(* IEC 61131-3 sources: matiec/tests/upstream_fixes, 6 files *)

(* ---- array_initializer_overflow.st ---- *)
(* Regression test for c73c55d (beremiz/matiec): too many initial values for
 * an array used to reach generate_c_vardecl.cc and hit an internal compiler
 * error instead of being caught in stage 3.
 *
 * c73c55d alone is not enough: its check reads symbol->datatype off the
 * array_initial_elements_list_c node, which is only ever set by 5b9968b ("Fix
 * initialization of arrays of non-simple types" -- it adds the
 * fill_candidate_datatypes_c/narrow_candidate_datatypes_c visitors for that
 * node). Without 5b9968b this test still reaches the same internal compiler
 * error, just as before c73c55d -- discovered while writing this test.
 *
 * Requires -p (forward references), since int_arr_t is used in the same file.
 *
 * Expect: a clean stage-3 error ("Too many initial values for array"),
 * exit != 0, and specifically NOT "Internal compiler error".
 *)
TYPE
  int_arr_t : ARRAY[0..1] OF INT;
END_TYPE

PROGRAM prog0
  VAR
    arr : int_arr_t := [1,2,3];
  END_VAR
  arr[0] := arr[0];
END_PROGRAM

CONFIGURATION config
  RESOURCE res ON PLC
    TASK tsk(INTERVAL := T#100ms, PRIORITY := 0);
    PROGRAM inst0 WITH tsk : prog0;
  END_RESOURCE
END_CONFIGURATION

(* ---- enum_in_array_initializer.st ---- *)
(* Regression test for f7185c6, exercising the array_spec_init_c path (rather
 * than initialized_structure_c) and depending on 5b9968b (see
 * array_initializer_overflow.st) to reach codegen at all: without 5b9968b,
 * narrow_candidate_datatypes_c never assigns a datatype to the
 * array_initial_elements_list_c node, and this crashes downstream in
 * generate_c_base.cc instead of exercising f7185c6's fix.
 *
 * Requires -p (forward references).
 *
 * Expect: clean compile, exit 0.
 *)
TYPE
  color_t : (RED, GREEN, BLUE);
END_TYPE

PROGRAM prog0
  VAR
    colors : ARRAY[0..2] OF color_t := [RED, GREEN, BLUE];
  END_VAR
  colors[0] := colors[0];
END_PROGRAM

CONFIGURATION config
  RESOURCE res ON PLC
    TASK tsk(INTERVAL := T#100ms, PRIORITY := 0);
    PROGRAM inst0 WITH tsk : prog0;
  END_RESOURCE
END_CONFIGURATION

(* ---- enum_in_struct_initializer.st ---- *)
(* Regression test for f7185c6 (beremiz/matiec): the stage3 enum-symtable
 * population visitors walked into aggregate initializer *values*, not just
 * their *specifications*, and crashed treating a referenced enum value
 * (RED, here) as if it were declaring a new one.
 *
 * Requires -p (forward references) since the STRUCT type is used the same file.
 *
 * Expect: clean compile, exit 0.
 *)
TYPE
  color_t : (RED, GREEN, BLUE);
  my_struct : STRUCT
    c : color_t;
  END_STRUCT;
END_TYPE

PROGRAM prog0
  VAR
    s : my_struct := (c := RED);
  END_VAR
  s.c := s.c;
END_PROGRAM

CONFIGURATION config
  RESOURCE res ON PLC
    TASK tsk(INTERVAL := T#100ms, PRIORITY := 0);
    PROGRAM inst0 WITH tsk : prog0;
  END_RESOURCE
END_CONFIGURATION

(* ---- f_trig_init.st ---- *)
(* Functional regression test for b082b44 / b3df950 (thiagoralves/matiec,
 * f-trigger-fix branch): F_TRIG's internal memory M was seeded FALSE. Since
 * F_TRIG_body__() computes Q := !CLK && !M *before* updating M := !CLK, an M
 * of FALSE means the very first evaluation with CLK still at its IEC-mandated
 * initial value of FALSE reports Q = TRUE -- a spurious trigger with no
 * preceding rising edge. M seeded TRUE fixes this (see f_trig_main.c, which
 * actually runs the compiled cycle and checks Q).
 *)
PROGRAM prog0
  VAR
    trig : F_TRIG;
    clk_in : BOOL := FALSE;
  END_VAR
  VAR_EXTERNAL
    q_out : BOOL;
  END_VAR
  trig(CLK := clk_in);
  q_out := trig.Q;
END_PROGRAM

CONFIGURATION config
  VAR_GLOBAL
    q_out : BOOL;
  END_VAR
  RESOURCE res ON PLC
    TASK tsk(INTERVAL := T#100ms, PRIORITY := 0);
    PROGRAM inst0 WITH tsk : prog0;
  END_RESOURCE
END_CONFIGURATION

(* ---- retain_shared_global.st ---- *)
(* Regression test for 12e4828 (beremiz/matiec): the per-name loop in
 * global_var_list_c::visit() reset current_varqualifier to none_vq after emitting
 * the first global of a shared VAR_GLOBAL RETAIN block, so every global after the
 * first fell back to print_retain()'s "retain" branch -- the literal identifier
 * `retain`, which config_init__() defines as 0 -- silently losing RETAIN.
 *
 * Expect: every one of g1, g2, g3 generates __INIT_GLOBAL(..., 1) in config.c,
 * not just g1.
 *)
PROGRAM prog0
  VAR
    x : INT;
  END_VAR
  x := 1;
END_PROGRAM

CONFIGURATION config
  VAR_GLOBAL RETAIN
    g1, g2, g3 : INT;
  END_VAR
  RESOURCE res ON PLC
    TASK tsk(INTERVAL := T#100ms, PRIORITY := 0);
    PROGRAM inst0 WITH tsk : prog0;
  END_RESOURCE
END_CONFIGURATION

(* ---- struct_initializer_member_order.st ---- *)
(* Regression test for c1df93e (beremiz/matiec): list_c::find_element() used
 * nocasecmp_c (a strict-weak "less than" functor) as an equality test. !ncc(a,b)
 * actually means a >= b, so the lookup returned the first member that sorts
 * alphabetically at-or-after the target name, instead of the exact match.
 *
 * "b" is declared before "a" here specifically to trigger the bug: looking up
 * "a" would incorrectly stop at "b" (the first element, which sorts after "a").
 *
 * IMPORTANT: this lookup is used for datatype-compatibility checking of the
 * initializer value, not for choosing which field the value is written to in
 * codegen (that goes through structure_element_name directly, unaffected by
 * this bug) -- a fixture with same-typed fields will compile "correctly" by
 * accident both with and without the fix, and prove nothing. b and a are
 * given deliberately incompatible types (STRING vs INT) so the bug produces
 * an observable false "incompatible datatype" error: with the bug, "a := 5"
 * gets checked against b's type (STRING) instead of a's (INT).
 *
 * Expect: clean compile, exit 0 (before the fix: a false datatype error).
 *)
TYPE
  my_struct : STRUCT
    b : STRING;
    a : INT;
  END_STRUCT;
END_TYPE

PROGRAM prog0
  VAR
    s : my_struct := (a := 5, b := 'hi');
  END_VAR
  s.a := s.a;
END_PROGRAM

CONFIGURATION config
  RESOURCE res ON PLC
    TASK tsk(INTERVAL := T#100ms, PRIORITY := 0);
    PROGRAM inst0 WITH tsk : prog0;
  END_RESOURCE
END_CONFIGURATION
